(* PLC project Tc2_System.GETCPUCOUNTER Demo, tc3-libraries-kb TwinCAT 3.1 *)
(* stored: creationDateTime 2026-05-20T00:00:00, modificationDateTime 2026-05-20T00:00:00 *)

PROGRAM P_Demo_GETCPUCOUNTER
  VAR
    fbGETCPUCOUNTER : GETCPUCOUNTER;  (* GETCPUCOUNTER 实例 *)
    udwCntLo : UDINT;  (* 64-bit 低 32 位 *)
    udwCntHi : UDINT;  (* 64-bit 高 32 位 *)
    ulCntCombined : ULINT;  (* 拼成 64-bit *)
  END_VAR

// ============================================================
// Tc2_System.GETCPUCOUNTER 演示程序
// ============================================================
// 场景：给工件打 100 ns 精度时间戳；24h 连续运行用 64-bit 不回卷。
// 价值：替代 F_GetSystemTime（NTP 同步会跳）。
// 验证：登录后 ulCntCombined 应持续单调递增，每个 PLC 周期增长约 (任务周期 / 100ns)。
// 验证步骤：
//   1. 右键 PLC 项目 → Import PLCopenXML → 选本文件
//   2. 引用 Tc2_System（References → Add library）
//   3. 编译 → 登录 → 运行；按上方『验证』指引在线写值观察
// ============================================================

fbGETCPUCOUNTER(cpuCntLoDW => udwCntLo, cpuCntHiDW => udwCntHi);

// 拼成 64-bit
ulCntCombined := SHL(TO_ULINT(udwCntHi), 32) OR TO_ULINT(udwCntLo);
END_PROGRAM
